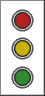
VISUALIZATION TrafficLight  // 45x96
VAR_IN_OUT
	Red : BOOL;
	Yellow : BOOL;
	Green : BOOL;
END_VAR
    Group (0,0 45x96)
        Rectangle (0,0 45x96)
        Lamp1 (10,8 25x25), variable: Red, style: Lamp-Lamp1-Red
        Lamp1 (10,36 25x25), variable: Yellow, style: Lamp-Lamp1-Yellow
        Lamp1 (10,65 25x25), variable: Green, style: Lamp-Lamp1-Green
END_VISUALIZATION

(* stored: Version 1.1.0.1
   Visu TrafficLight: Id {e733daa0-66b7-44dd-b113-4b2ccd3a5ba7} *)
